// TIA Portal V18 export
DATA_BLOCK "VirtModulesConf"   // DB10003
{ S7_Optimized_Access := 'FALSE' }
VERSION : 0.1
// stored: AutoNumber false, DBAccessibleFromOPCUA true, IsOnlyStoredInLoadMemory false, IsWriteProtectedInAS false
   VAR
      Virt { S7_SetPoint := 'True'} : Array[1..4] of "UDT_VirtModulesMap";
   END_VAR
BEGIN
   Virt[1..4].cRack := 111;
   Virt[1].cModule := 1;
   Virt[2].cModule := 2;
   Virt[3].cModule := 3;
   Virt[4].cModule := 4;
END_DATA_BLOCK
